// TIA Portal V16 export
// export: Created 2021-07-12T14:47:17.796924Z, ExportSetting WithDefaults, DisplayName Totally Integrated Automation Portal, DisplayVersion V16, DisplayName TIA Portal Version Control Interface, DisplayVersion V16, DisplayName TIA Portal Openness, DisplayVersion V16, DisplayName STEP 7 Professional, DisplayVersion V16, DisplayName STEP 7 Safety, DisplayVersion V16, DisplayName WinCC Professional, DisplayVersion V16
TYPE "LSimaHydTO_typeMotionVector"
TITLE = LSimaHydTO_typeMotionVector
// Values of a motion vector
// stored: IsFailsafeCompliant false
   STRUCT
      Position : LReal;   // Position
      Velocity : LReal;   // Velocity
      Acceleration : LReal;   // Acceleration
   END_STRUCT;
END_TYPE
